// Mitsubishi GX Works2 project: part2   PLC: FX3G

// global labels: Global1
VAR_GLOBAL
  HeatSpreader_on AT Y000 : BOOL;
  switchStart AT X001 : BOOL;
  temp_above25 AT X003 : BOOL;
  heaterDiffuser AT Y007 : BOOL;
  temp_lower20 AT X002 : BOOL;
  temp_lower30 AT X004 : BOOL;
  TC AT TC30 : BOOL;
END_VAR
VAR_GLOBAL CONSTANT
  FiveSec : REAL := 50;
END_VAR
VAR_GLOBAL
  Lamp AT Y010 : BOOL;
END_VAR

// task Task_01 (event TRUE, interval 0, priority 31): POU_01

PROGRAM POU_01
(* structured ladder/FBD written out as ST: instructions are called as NAME(EN, inputs, outputs); _pN, _eN, _tN stand for wires *)
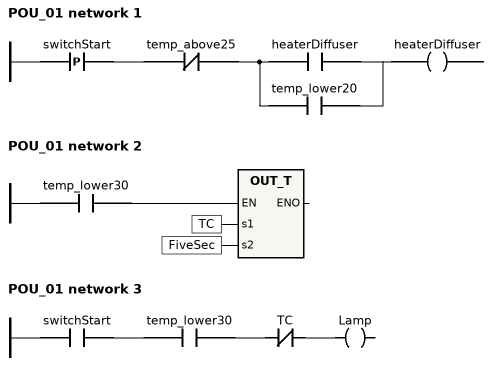
(* network 1 *)
_p1 := LDP(TRUE, switchStart) AND NOT temp_above25;
heaterDiffuser := (_p1 AND heaterDiffuser) OR (_p1 AND temp_lower20);
(* network 2 *)
OUT_T(temp_lower30, TC, FiveSec);
(* network 3 *)
Lamp := switchStart AND temp_lower30 AND NOT TC;
END_PROGRAM
